TYPE OutMotorCommands :
STRUCT
	controlword: UINT;
	target_positon: DINT;
	motor_op_out: SINT;
	profile_vel: UDINT;
	profile_accel: UDINT;
	profile_decel: UDINT;
END_STRUCT
END_TYPE

(* stored: Version 1.1.0.1, ProductVersion 3.1.4024.12
   DUT OutMotorCommands: Id {618dcf93-122c-48c9-8754-57ce26939a3c} *)
